TYPE ST_RecipeTypeLeakTestStep :
STRUCT
	nIdx	: UINT;
	bEnable	: BOOL;
	nActiveSubStepCount		: UINT; // Default 0; No Sub Step Exist
	nValveMaskForThisStep	: UDINT; // Debug; ULINT 64 bit cannot be saved on TcHmi; Data REGEX type does not Match check with support
	bApplyTimeOffDelay	: BOOL;
	bApplyTimeOnDelay	: BOOL;
	tTimeOffDelay	: TIME;
	tTimeOnDelay	: TIME;
END_STRUCT
END_TYPE

(* stored: Version 1.1.0.1
   DUT ST_RecipeTypeLeakTestStep: Id {8d086e50-fc40-0b38-27ae-4d07d08c84e7} *)
